TYPE E_PalletOrientation :
(
	OrientationZero,
	OrientationNinty,
	OrientationOneEighty,
	OrientationTwoSeventy
);
END_TYPE

(* stored: Version 1.1.0.1, ProductVersion 3.1.4022.12
   DUT E_PalletOrientation: Id {350541a7-ea79-4386-9754-b4efb965bd56} *)
